TYPE ST_TransportTube :
STRUCT
	sName : STRING(10);
	stDevices : ST_TransportTubeDevices;
END_STRUCT
END_TYPE

(* stored: Version 1.1.0.1, ProductVersion 3.1.4022.17
   DUT ST_TransportTube: Id {8992122d-47b4-43be-a476-1a9903008ec1} *)
